ABB RobotStudio station: Station.rsstn

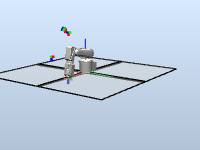
Station Station (saved by RobotStudio 6.5.7502.1049)
Controller MTRN4230
  mechanical unit ROB_1: IRB120_3_58__01, 6 joints, base frame (0, 0, 0) mm
Layout (positions relative to the parent item):
  - IRB120_3_58__01 [mechanism, from Robots\IRB120_3_58_G_01.rslib] at (0, 0, 0) mm; joint values [0.0108, 1.3982, 0, 0, 0, 0] (rad or m)
Collision set CollisionSet_1:  against , near miss 0.003 m
Targets, tools, work objects and paths stored in the station, written as RAPID:
! task T_ROB1
MODULE Module1
  CONST robtarget Target_10:=[[0.000028236,-374,630],[0.500000019,0.499999981,0.500000019,-0.499999981],[-1,0,0,0],[9E+09,9E+09,9E+09,9E+09,9E+09,9E+09]];
  CONST robtarget Target_20:=[[0.000029797,-394.667942477,605.773993832],[0.433593745,0.461814156,0.564103961,-0.52963277],[-1,-1,0,1],[9E+09,9E+09,9E+09,9E+09,9E+09,9E+09]];
  CONST robtarget Target_30:=[[0.000029797,-394.667942477,605.773993832],[0.433593745,0.461814156,0.564103961,-0.52963277],[-1,0,-1,0],[9E+09,9E+09,9E+09,9E+09,9E+09,9E+09]];
  CONST jointtarget JointTarget_3:=[[0,0,0,0,0,0],[9E+09,9E+09,9E+09,9E+09,9E+09,9E+09]];
  CONST robtarget Target_40:=[[174.884571922,-518.218749422,206.781458264],[0.005358512,-0.583622229,-0.811993821,-0.004734365],[-1,0,0,0],[9E+09,9E+09,9E+09,9E+09,9E+09,9E+09]];
  PROC Path_10()
  ENDPROC
ENDMODULE

